TYPE ZData :
STRUCT
  Config : ZDataConfig;
  Machine : ZDataMachine;
  Calibration : ZDataCalibration;
  Recipe : ZDataRecipe;
END_STRUCT
END_TYPE

(* stored: Version 1.1.0.1
   DUT ZData: Id {6b0931f8-773c-4ef9-8596-c6964545b443} *)
